// TIA Portal V17 export
// export: Created 2025-03-10T12:14:37.2684978Z, ExportSetting WithDefaults, DisplayName Totally Integrated Automation Portal, DisplayVersion V17 Update 8, DisplayName TIA Portal Openness, DisplayVersion V17 Update 8, DisplayName TIA Portal Version Control Interface, DisplayVersion V17, DisplayName SINAMICS Startdrive Advanced, DisplayVersion V17 SP2, DisplayName SINAMICS Startdrive G110M, G120, G120C, G120D, G120P, G115D, DisplayVersion V17 SP2, DisplayName SINAMICS Startdrive G130, G150, S120, S150, SINAMICS MV, S210, DisplayVersion V17 SP2, DisplayName STEP 7 Professional, DisplayVersion V17 Update 8, DisplayName SINUMERIK ONE STEP 7 Toolbox, DisplayVersion V17 Update 12, DisplayName SINUMERIK 840D sl STEP 7 Toolbox, DisplayVersion V17 Update 12, DisplayName STEP 7 Safety, DisplayVersion V17 Update 6, DisplayName WinCC Advanced, DisplayVersion V17 Update 8
DATA_BLOCK "LBP_TMTurret"   // DB73
TITLE = Tool management / Gestión de herramientas / Werkzeugverwaltung
{ S7_Optimized_Access := 'FALSE'; DB_Accessible_From_OPC_UA := 'FALSE' }
AUTHOR : SINUMERIK
FAMILY : SINUMERIK_ONE
VERSION : 6.15
// Interface between user program and tool management, contains signals for turret. / Interfaz entre programa de usuario y gestión de herramientas, contiene señales para torreta/revólver / Schnittstelle zwischen Anwenderprogramm und Werkzeugverwaltung, enthält Signale für Revolver
// stored: AutoNumber false, DBAccessibleFromOPCUA false, DBAccessibleFromWebserver true, InstanceOfName LBP_typeTMTurret, InstanceOfType UDT, IsOnlyStoredInLoadMemory false, IsWriteProtectedInAS false
"LBP_typeTMTurret"
   // VAR RETAIN
   //    IFNo : Array[1..16] of Bool;
   //    Quit : Array[1..16] of Bool;
   //    TIF : Array[1..16] of Struct
   //       Comp : Bool;
   //       Perform : Bool;
   //       f0_2 : Bool;
   //       T0 : Bool;
   //       f0_4 : Bool;
   //       f0_5 : Bool;
   //       ManTOut : Bool;
   //       f0_7 : Bool;
   //       PerfStatusError : Bool;
   //       n1_1 : Bool;
   //       n1_2 : Bool;
   //       n1_3 : Bool;
   //       n1_4 : Bool;
   //       n1_5 : Bool;
   //       n1_6 : Bool;
   //       DataInDB1073 : Bool;
   //       Channel : Byte;
   //       TMNo : Byte;
   //       VdiTcp0 : DInt;
   //       VdiTcp1 : DInt;
   //       VdiTcp2 : DInt;
   //       BufferIdent : Int;
   //       BufferNo : Int;
   //       SMag : Int;
   //       SLoc : Int;
   //       TMag : Int;
   //       TLoc : Int;
   //       LocType : Int;
   //       SLeft : Int;
   //       SRight : Int;
   //       STop : Int;
   //       SBottom : Int;
   //       TInBuffer : Bool;
   //       IgnoreDisabled : Bool;
   //       Unload : Bool;
   //       Load : Bool;
   //       MasterTool : Bool;
   //       n38_5 : Bool;
   //       Exchange_1to1 : Bool;
   //       HandTool : Bool;
   //       Active : Bool;
   //       Enabled : Bool;
   //       Disabled : Bool;
   //       Measured : Bool;
   //       Prewarn : Bool;
   //       Change : Bool;
   //       FixedLoc : Bool;
   //       Used : Bool;
   //       TNo : Int;
   //       MyPlace : Int;
   //    END_STRUCT;
   // END_VAR
BEGIN
END_DATA_BLOCK
